// SIMATIC S7-200 SMART project (STEP 7-Micro/WIN SMART), CPU ST40

SYMBOL_TABLE Table 1
Item_detected    V0.0
Lid_at_place     V0.1
Base_at_place    V0.2
Part_leaving     V0.3
Start            V0.4
Reset            V0.5
Stop_            V0.6
Emergency_stop   V0.7
Auto             V1.0
FACTORY_IO_Running V1.1
X                VD100
Z                VD104
Lids_conveyor_1  Q0.0
Stop_blade_1     Q0.1
Lids_conveyor_2  Q0.2
Bases_conveyor_1 Q0.3
Stop_blade_2     Q0.4
Bases_conveyor_2 Q0.5
Grab             Q0.6
Start_light      Q0.7
Reset_light      Q1.0
Stop_light       Q1.1
Set_X            QD4
Set_Z            QD8
Counter          QD12
END_SYMBOL_TABLE

SYMBOL_TABLE System Symbols
Always_On        SM0.0    // Always ON
END_SYMBOL_TABLE

ORGANIZATION_BLOCK MAIN:OB1
TITLE=Program Comments
BEGIN
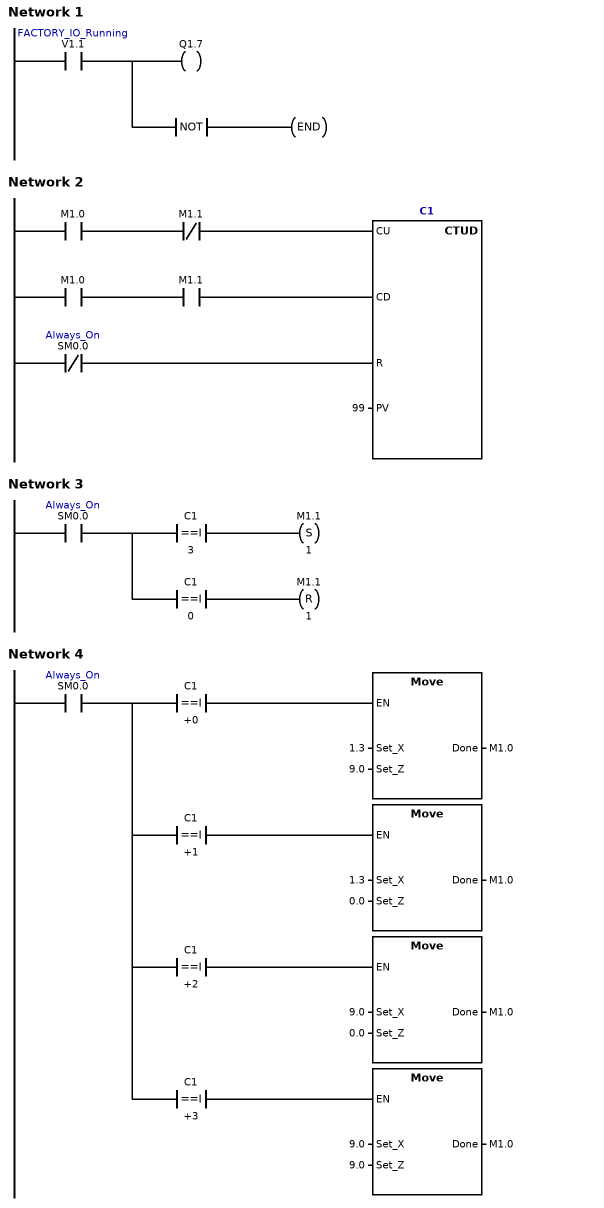
Network 1
LD     FACTORY_IO_Running:V1.1
=      Q1.7
NOT
END
Network 2
LD     M1.0
AN     M1.1
LD     M1.0
A      M1.1
LDN    Always_On:SM0.0
CTUD   C1, 99
Network 3
LD     Always_On:SM0.0
LPS
AW=    C1, 3
S      M1.1, 1
LPP
AW=    C1, 0
R      M1.1, 1
Network 4
LD     Always_On:SM0.0
LPS
AW=    C1, +0
CALL   Move:SBR0, 1.3, 9.0, M1.0
LRD
AW=    C1, +1
CALL   Move:SBR0, 1.3, 0.0, M1.0
LRD
AW=    C1, +2
CALL   Move:SBR0, 9.0, 0.0, M1.0
LPP
AW=    C1, +3
CALL   Move:SBR0, 9.0, 9.0, M1.0
END_ORGANIZATION_BLOCK

SUBROUTINE_BLOCK Move:SBR0
TITLE=Subroutine Comments
VAR_INPUT
Set_X:REAL;	// LD0 
Set_Z:REAL;	// LD4 
END_VAR
VAR_OUTPUT
Done:BOOL;	// L8.0 
END_VAR
VAR
tmp:BOOL;	// L8.1 
tmp_x:REAL;	// LD9 
tmp_z:REAL;	// LD13 
END_VAR
BEGIN
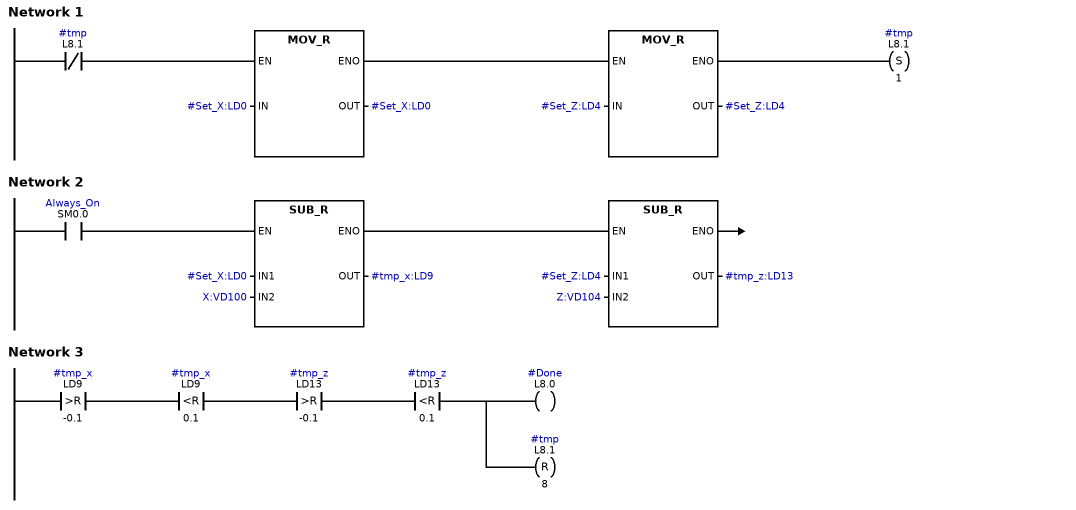
Network 1
LDN    #tmp:L8.1
MOVR   #Set_X:LD0, Set_X:QD4
AENO
MOVR   #Set_Z:LD4, Set_Z:QD8
AENO
S      #tmp:L8.1, 1
Network 2
// (network saved uncompiled; LAD cells follow)
// row 0: c0 -| |- Always_On:SM0.0  c1 --  c2 [SUB_R EN:=power@row0, IN1:=#Set_X:LD0, IN2:=X:VD100, ENO=>power, OUT=>#tmp_x:LD9]  c3 --  c4 --  c5 [SUB_R EN:=power@row0, IN1:=#Set_Z:LD4, IN2:=Z:VD104, ENO=>power, OUT=>#tmp_z:LD13]  c6 ->
// row 1: c2 [box]  c5 [box]
Network 3
LDR>   #tmp_x:LD9, -0.1
AR<    #tmp_x:LD9, 0.1
AR>    #tmp_z:LD13, -0.1
AR<    #tmp_z:LD13, 0.1
=      #Done:L8.0
R      #tmp:L8.1, 8
END_SUBROUTINE_BLOCK

// SBR1: protected block, not included

// SBR2: protected block, not included
